FUNCTION_BLOCK Profesor EXTENDS Persona IMPLEMENTS ITF_Profesor
VAR_INPUT
END_VAR
VAR_OUTPUT
END_VAR
VAR
	_Nombre: STRING;
END_VAR

METHOD DarClases
VAR_INPUT
END_VAR
END_METHOD

{warning 'Agregar implementación de método'}
METHOD Fichar
END_METHOD

PROPERTY Nombre : String
GET
END_GET
SET
END_SET
END_PROPERTY

{warning 'Agregar implementación de propiedad'}
PROPERTY Salida : INT
GET
END_GET
SET
END_SET
END_PROPERTY

END_FUNCTION_BLOCK

(* stored: Version 1.1.0.1, ProductVersion 3.1.4024.12
   POU Profesor: Id {b7884ec5-07e8-4a6e-9269-8fa6a6554ecf}, SpecialFunc None
   Method DarClases: Id {6b209387-2537-402c-81fd-921a69adf89b}
   Method Fichar: Id {f9336cb5-f090-43e7-b6db-0621fc018b38}
   Property Nombre: Id {17598f38-9bdf-45fe-9441-8725ae07811a}
   Get Get: Id {87b041bc-6822-43ec-93ad-c40b1360a8ff}
   Set Set: Id {e220a405-94dc-4330-b6e9-48301bcf83cf}
   Property Salida: Id {faf22ff7-7886-4e56-8833-347250fbf2c2}
   Get Get: Id {f6a5a615-9366-45bd-ba8d-e9f12554731e}
   Set Set: Id {bca320ab-790c-4e80-90bd-4a763e48037e} *)
